(* CODESYS project GVL.export

Project tree, tasks and I/O mapping:
  global variables GVL
*)

// GVL
{attribute 'qualified_only'}
VAR_GLOBAL
	(**** OPERATION MODE ****)
	Inititialisation_OK	 :BOOL;
	Auto	:BOOL;
	Auto_Stop	:BOOL;
	Auto_Run :BOOL;
	E_Stop	: BOOL;
	Manual	:BOOL;
	Confirmation_Required	:BOOL;
	blinker : TON;
	flash : BOOL;
END_VAR
